TYPE ST_DefectTable :
STRUCT
	InstancePath: T_InstancePath;
	Description: STRING;
	State: E_DefectState;
	Severity: TcEventSeverity;
	ErrorID: STRING(3);
	ClassID: STRING(3);
	Color: DWORD;
	RisingEdge: T_MaxString;
	FallingEdge: T_MaxString;
END_STRUCT
END_TYPE

(* stored: Version 1.1.0.1, ProductVersion 3.1.4024.12
   DUT ST_DefectTable: Id {cf38894e-519c-4c1d-85d5-079b920fd2fe} *)
